FUNCTION_BLOCK fb_gm_measurementModule
VAR_INPUT
	SFCInit : BOOL;
END_VAR
VAR_OUTPUT
END_VAR
VAR
	trn_connectionCheckDone: BOOL;
	trn_wattingForLensDone: BOOL;
	flg_buf_gateLengthISSuccessed: BOOL;
	flg_buf_dummySignal: BOOL;
	trn_readCavDone: BOOL;
	fbi_getCav: fb_getCav;
	trn_chuckDone: BOOL;
	var_chuckCount: INT;
	trn_requestPickUpDone: BOOL;
	TON_data: TON;
	fbi_delayTimer: TON;
	trn_AddCountDone: BOOL;
	trn_lotStampDone: BOOL;
	var_process: INT;
	fbi_ton: TON;
	trn_LensCheckDone: BOOL;
	flg_SensorCheckDone: BOOL;
	flg_incjet_runned: BOOL;
END_VAR

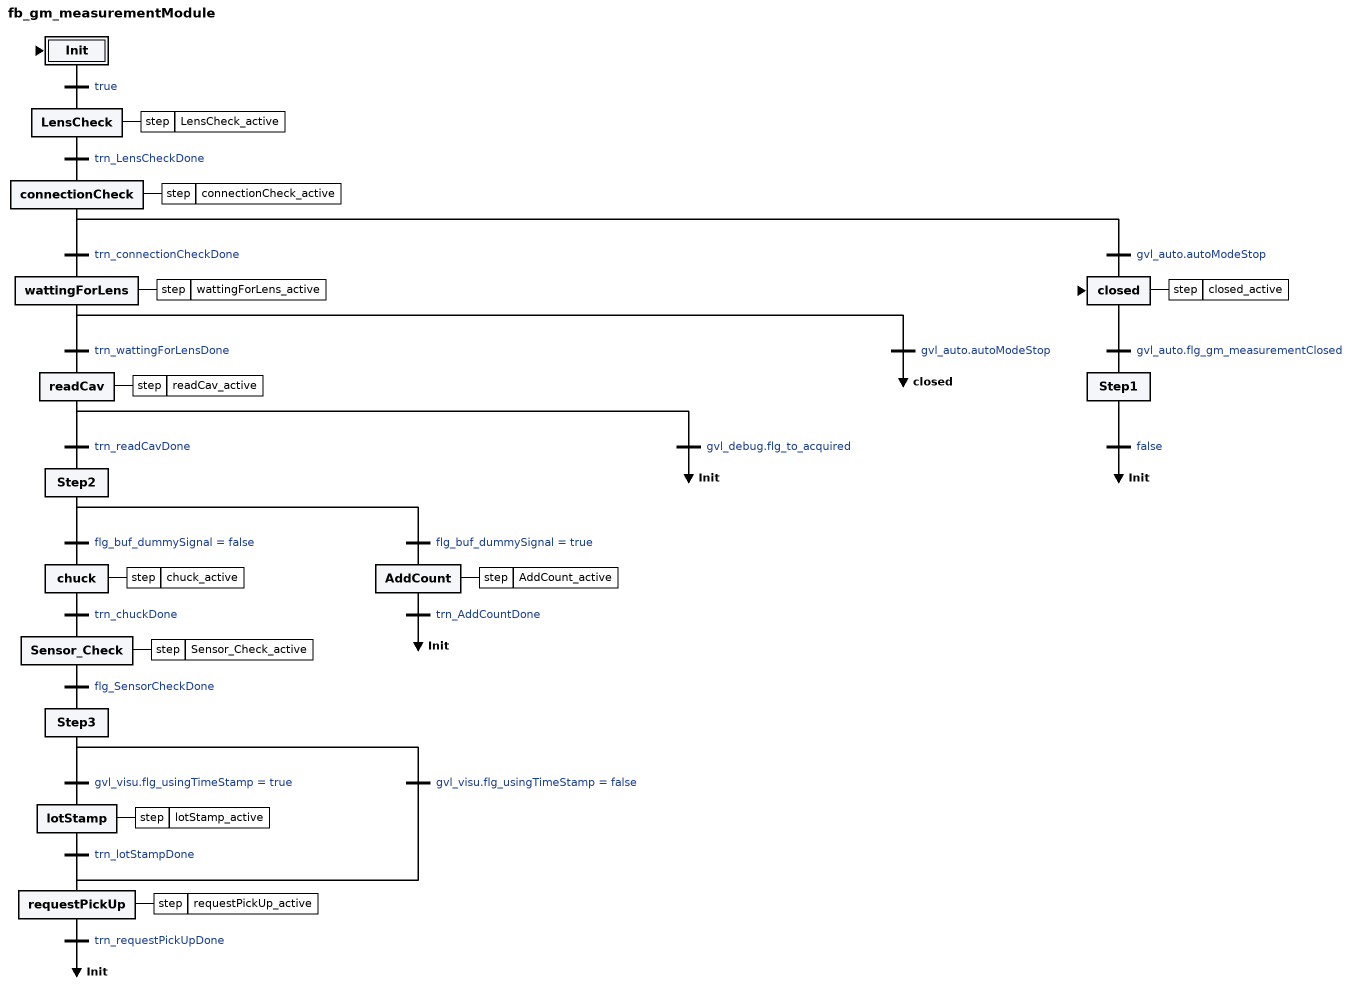
INITIAL_STEP Init:
END_STEP
TRANSITION FROM Init TO LensCheck
    := true;
END_TRANSITION
STEP LensCheck:
    LensCheck_active(N);  // step action
END_STEP
TRANSITION FROM LensCheck TO connectionCheck
    := trn_LensCheckDone;
END_TRANSITION
STEP connectionCheck:
    connectionCheck_active(N);  // step action
END_STEP
TRANSITION FROM connectionCheck TO wattingForLens
    := trn_connectionCheckDone;
END_TRANSITION
STEP wattingForLens:
    wattingForLens_active(N);  // step action
END_STEP
TRANSITION FROM wattingForLens TO readCav
    := trn_wattingForLensDone;
END_TRANSITION
TRANSITION FROM wattingForLens TO closed
    := gvl_auto.autoModeStop;
END_TRANSITION
TRANSITION FROM connectionCheck TO closed
    := gvl_auto.autoModeStop;
END_TRANSITION
STEP closed:
    closed_active(N);  // step action
END_STEP
TRANSITION FROM closed TO Step1
    := gvl_auto.flg_gm_measurementClosed;
END_TRANSITION
STEP Step1:
END_STEP
TRANSITION FROM Step1 TO Init
    := false;
END_TRANSITION
STEP readCav:
    readCav_active(N);  // step action
END_STEP
TRANSITION FROM readCav TO Step2
    := trn_readCavDone;
END_TRANSITION
TRANSITION FROM readCav TO Init
    := gvl_debug.flg_to_acquired;
END_TRANSITION
STEP Step2:
END_STEP
TRANSITION FROM Step2 TO chuck
    := flg_buf_dummySignal = false;
END_TRANSITION
TRANSITION FROM Step2 TO AddCount
    := flg_buf_dummySignal = true;
END_TRANSITION
STEP AddCount:
    AddCount_active(N);  // step action
END_STEP
TRANSITION FROM AddCount TO Init
    := trn_AddCountDone;
END_TRANSITION
STEP chuck:
    chuck_active(N);  // step action
END_STEP
TRANSITION FROM chuck TO Sensor_Check
    := trn_chuckDone;
END_TRANSITION
STEP Sensor_Check:
    Sensor_Check_active(N);  // step action
END_STEP
TRANSITION FROM Sensor_Check TO Step3
    := flg_SensorCheckDone;
END_TRANSITION
STEP Step3:
END_STEP
TRANSITION FROM Step3 TO lotStamp
    := gvl_visu.flg_usingTimeStamp = true;
END_TRANSITION
STEP lotStamp:
    lotStamp_active(N);  // step action
END_STEP
TRANSITION FROM lotStamp TO requestPickUp
    := trn_lotStampDone;
END_TRANSITION
TRANSITION FROM Step3 TO requestPickUp
    := gvl_visu.flg_usingTimeStamp = false;
END_TRANSITION
STEP requestPickUp:
    requestPickUp_active(N);  // step action
END_STEP
TRANSITION FROM requestPickUp TO Init
    := trn_requestPickUpDone;
END_TRANSITION

ACTION AddCount_active:
IF AddCount._x AND AddCount.x = FALSE THEN
	trn_AddCountDone := FALSE;
ELSIF AddCount._x AND AddCount.x THEN
	IF gvl_visu.flg_missingParts THEN
		gvl_gm.var_buf_measurementCav := gvl_auto.pocketNo[gvl_auto.buf_cavNo] + 1;
		trn_AddCountDone := TRUE;
	ELSE
		trn_AddCountDone := TRUE;
	END_IF
END_IF
END_ACTION

ACTION chuck_active:
IF chuck._x AND chuck.x = FALSE THEN
	TON_data.IN := FALSE;;
	trn_chuckDone := FALSE;
	gvl_solv.fbi_gm_chuck.in_flg_run := FALSE;
	gvl_solv.fbi_gm_push.in_flg_run := FALSE;
	gvl_auto.flg_gateData_Tx := FALSE;
	var_chuckCount := -11;
ELSIF chuck._x AND chuck.x THEN
	CASE var_chuckCount OF
		-11:
			IF gvl_param.var_productInfo[gvl_param.var_currentProductID].flg_mode_measurement THEN
				var_chuckCount := -10;
			ELSE
				var_chuckCount := 0;
			END_IF
		-10:
			gvl_solv.fbi_gm_push.in_var_moveMode := eP_svMoveMode.svB;
			gvl_solv.fbi_gm_push.in_flg_run := TRUE;
			var_chuckCount := -9;
		-9:
			IF gvl_solv.fbi_gm_push.out_flg_Done THEN
				gvl_solv.fbi_gm_push.in_flg_run := FALSE;
				var_chuckCount := -8;
			END_IF
		-8:
			gvl_solv.fbi_gm_push.in_var_moveMode := eP_svMoveMode.svA;
			gvl_solv.fbi_gm_push.in_flg_run := TRUE;
			var_chuckCount := -7;
		-7:
			IF gvl_solv.fbi_gm_push.out_flg_Done THEN
				gvl_solv.fbi_gm_push.in_flg_run := FALSE;
				var_chuckCount := -6;
			END_IF
		-6:
			gvl_solv.fbi_gm_chuck.in_var_moveMode := eP_svMoveMode.svB;
			gvl_solv.fbi_gm_chuck.in_flg_run := TRUE;
			var_chuckCount := -5;
		-5:
			IF gvl_solv.fbi_gm_chuck.out_flg_Done THEN
				gvl_solv.fbi_gm_chuck.in_flg_run := FALSE;
				var_chuckCount := -4;
			END_IF
		-4:
			gvl_solv.fbi_gm_push.in_var_moveMode := eP_svMoveMode.svB;
			gvl_solv.fbi_gm_push.in_flg_run := TRUE;
			var_chuckCount := -3;
		-3:
			IF gvl_solv.fbi_gm_push.out_flg_Done THEN
				gvl_solv.fbi_gm_push.in_flg_run := FALSE;
				var_chuckCount := 6;
			END_IF
		0:
			gvl_solv.fbi_gm_chuck.in_var_moveMode := eP_svMoveMode.svB;
			gvl_solv.fbi_gm_chuck.in_flg_run := TRUE;
			var_chuckCount := 1;
		1:
			
			IF gvl_solv.fbi_gm_chuck.out_flg_Done THEN
				gvl_solv.fbi_gm_chuck.in_flg_run := FALSE;
				var_chuckCount := 2;
			END_IF
		2:
			
			gvl_solv.fbi_gm_chuck.in_var_moveMode := eP_svMoveMode.svA;
			gvl_solv.fbi_gm_push.in_var_moveMode := eP_svMoveMode.svB;
			gvl_solv.fbi_gm_push.in_flg_run := TRUE;
			gvl_solv.fbi_gm_chuck.in_flg_run := TRUE;
			var_chuckCount := 3;
		3:
			IF gvl_solv.fbi_gm_push.out_flg_Done THEN
				gvl_solv.fbi_gm_push.in_flg_run := FALSE;
				gvl_solv.fbi_gm_chuck.in_flg_run := FALSE;
				var_chuckCount := 4;
			END_IF
		4:
			gvl_solv.fbi_gm_chuck.in_var_moveMode := eP_svMoveMode.svB;
			gvl_solv.fbi_gm_chuck.in_flg_run := TRUE;
			var_chuckCount := 5;
		5:
			IF gvl_solv.fbi_gm_chuck.out_flg_Done THEN
				gvl_solv.fbi_gm_chuck.in_flg_run := FALSE;
				var_chuckCount := 6;
			END_IF
		6:	
			TON_data.IN := TRUE;
			IF TON_data.Q THEN
				var_chuckCount := 7;
			END_IF
		7://gate measurement
			TON_data.IN := FALSE;
			IF gvl_io.flg_gm_fiberSens AND (gvl_io.var_gateLength > gvl_param.var_productInfo[gvl_param.var_currentProductID].gateLength_max OR gvl_io.var_gateLength < gvl_param.var_productInfo[gvl_param.var_currentProductID].gateLength_min) THEN
				gvl_gm.flg_gateLengthIsPassed := FALSE;
			ELSE
				gvl_gm.flg_gateLengthIsPassed := TRUE;
			END_IF
			gvl_auto.flg_gateData_Tx := TRUE;
			var_chuckCount := 8;
		8:
			gvl_solv.fbi_gm_chuck.in_flg_run := FALSE;
			var_chuckCount := 9;
		9:
			trn_chuckDone := TRUE;
	END_CASE
END_IF
TON_data(IN:= , PT:=T#200MS , Q=> , ET=> );
END_ACTION

ACTION closed_active:
IF closed._x AND closed.x = FALSE THEN
	gvl_auto.flg_gm_measurementClosed := FALSE;
ELSIF closed._x AND closed.x THEN
	gvl_io.flg_requestLens := FALSE;
	gvl_auto.flg_gm_measurementClosed := TRUE;
END_IF
END_ACTION

ACTION connectionCheck_active:
IF connectionCheck._x AND connectionCheck.x = FALSE THEN
	trn_connectionCheckDone:= FALSE;
	gvl_io.flg_requestLens := TRUE;
	var_process := 0;
ELSIF connectionCheck._x AND connectionCheck.x THEN
	CASE var_process OF
		0:
			IF gvl_io.flg_bitNumber0 
				AND gvl_io.flg_bitNumber1
				AND gvl_io.flg_bitNumber2
				AND gvl_io.flg_bitNumber3 OR gvl_debug.cavConecctSkip THEN
				trn_connectionCheckDone:= TRUE;
			END_IF
			IF NOT gvl_visu.flg_btn_vacSensOn THEN
				IF gvl_io.flg_gm_fiberSens THEN
					gvl_io.flg_requestLens := FALSE;
					IF((gvl_axis.axisX.NcToPlc.ActPos < gvl_visu.var_in_initialPos.x + 1) AND (gvl_axis.axisX.NcToPlc.ActPos > gvl_visu.var_in_initialPos.x - 1) AND NOT gvl_io.flg_fiberSens AND gvl_io.out_wire_ejectorVac ) THEN
						gvl_error.flg_gm_fiberSens := TRUE;
					END_IF
				END_IF
			END_IF
	END_CASE
	
END_IF
END_ACTION

ACTION LensCheck_active:
IF LensCheck._x AND LensCheck.x = FALSE THEN
	trn_LensCheckDone := FALSE;
	gvl_debug.flg_to_demand:= FALSE;
ELSIF LensCheck._x AND LensCheck.x THEN
	IF gvl_debug.out_busy THEN
		trn_LensCheckDone := TRUE;
	ELSE
		IF gvl_io.flg_gm_fiberSens THEN
			gvl_error.flg_gm_fiberSens := TRUE;	
		ELSE
			trn_LensCheckDone := TRUE;
		END_IF	
	END_IF
END_IF
END_ACTION

ACTION lotStamp_active:
IF lotStamp._x AND lotStamp.x = FALSE THEN
	trn_lotStampDone := FALSE;
	var_process := 0;
	fbi_ton.IN := FALSE;
	flg_incjet_runned:= FALSE;
ELSIF lotStamp._x AND lotStamp.x THEN
	CASE var_process OF
		0:
			fbi_ton.PT:= T#5S;
			fbi_ton.IN := TRUE;
			gvl_error.flg_incjet := fbi_ton.Q;
			gvl_gm.var_incjetInfo.flg_denyStamp := gvl_io.flg_gm_fiberSens;
			IF gvl_gm.var_incjetInfo.flg_stampReady THEN
				var_process := 1;
			END_IF
		1:
			fbi_ton.IN := FALSE;
			gvl_solv.fbi_gm_stamp.in_flg_run := FALSE;
			gvl_solv.fbi_gm_stamp.in_var_moveMode := eP_svMoveMode.svB;
			var_process := 2;
			
		2:
			gvl_solv.fbi_gm_stamp.in_flg_run := TRUE;
			var_process := 3;
		3:
			IF gvl_gm.var_incjetInfo.flg_stampRun THEN
				flg_incjet_runned:= TRUE;
			END_IF
			IF gvl_solv.fbi_gm_stamp.out_flg_Done THEN
				gvl_solv.fbi_gm_stamp.in_flg_run := FALSE;
				var_process := 4;
			END_IF
		4:
			fbi_ton.PT:= T#0.2S;
			fbi_ton.IN := TRUE;
			IF gvl_gm.var_incjetInfo.flg_stampRun THEN
				flg_incjet_runned:= TRUE;
			END_IF
			IF fbi_ton.Q THEN
				var_process := 5;
			END_IF
		5:
			IF flg_incjet_runned OR NOT gvl_gm.var_incjetInfo.flg_denyStamp THEN
				var_process := 6;
			ELSE
				gvl_error.flg_incjet:= TRUE;
			END_IF
		6:
			fbi_ton.IN := FALSE;
			gvl_solv.fbi_gm_stamp.in_var_moveMode := eP_svMoveMode.svA;
			gvl_solv.fbi_gm_stamp.in_flg_run := TRUE;
			var_process := 7;
		7:
			IF gvl_solv.fbi_gm_stamp.out_flg_Done THEN
				gvl_solv.fbi_gm_stamp.in_flg_run := FALSE;
				var_process := 8;
			END_IF
		8:
			flg_incjet_runned:= FALSE;
			gvl_gm.var_incjetInfo.flg_denyStamp := FALSE;
			trn_lotStampDone := TRUE;
	END_CASE
END_IF
fbi_ton(IN:= , PT:= , Q=> , ET=> );
END_ACTION

ACTION readCav_active:
IF readCav._x AND readCav.x = FALSE THEN
	trn_readCavDone := FALSE;
	THIS^.fbi_getCav();
	fbi_getCav.in_flg_run := FALSE;
	fbi_delayTimer.IN := FALSE;
ELSIF readCav._x AND readCav.x THEN
	THIS^.fbi_getCav();
	fbi_delayTimer.IN := TRUE;
	THIS^.fbi_getCav.in_flg_run := fbi_delayTimer.Q;
	IF gvl_debug.flg_debug_run THEN
		gvl_gm.var_buf_measurementCav := gvl_debug.var_cav;
		IF NOT (gvl_debug.flg_check_quality AND gvl_debug.flg_to_measurement) THEN
			trn_readCavDone := TRUE;
		END_IF
	ELSE
		IF THIS^.fbi_getCav.out_flg_Done THEN
			gvl_gm.var_buf_measurementCav := THIS^.fbi_getCav.out_var_cav;
			IF gvl_debug.flg_check_quality AND gvl_debug.flg_to_measurement THEN
				gvl_debug.flg_to_demand:= TRUE;
			ELSE
				trn_readCavDone := TRUE;
			END_IF
		ELSIF THIS^.fbi_getCav.out_flg_error THEN
			gvl_auto.cavNo := 0;
			IF gvl_debug.flg_check_quality AND gvl_debug.flg_to_measurement THEN
				gvl_debug.flg_to_demand:= TRUE;
			ELSE
				trn_readCavDone := TRUE;
			END_IF
		END_IF
	END_IF	
	
END_IF
fbi_delayTimer(IN:= , PT:=T#100MS , Q=> , ET=> );
END_ACTION

ACTION requestPickUp_active:
IF requestPickUp._x AND requestPickUp.x = FALSE THEN
	gvl_gm.flg_lensPickUpDone := FALSE;
	gvl_gm.flg_requestPickup := FALSE;
	trn_requestPickUpDone := false;
ELSIF requestPickUp._x AND requestPickUp.x THEN
	IF gvl_gm.flg_lensPickUpDone THEN
		gvl_gm.flg_requestPickup := FALSE;
		trn_requestPickUpDone := TRUE;
	ELSE
		gvl_gm.flg_requestPickup := TRUE;
	END_IF
END_IF
END_ACTION

ACTION Sensor_Check_active:
IF Sensor_Check._x AND Sensor_Check.x = FALSE THEN
	flg_SensorCheckDone := FALSE;
ELSIF Sensor_Check._x AND Sensor_Check.x THEN
	IF gvl_visu.flg_btn_vacSensOn THEN
		flg_SensorCheckDone:= TRUE;
	ELSE
		IF gvl_io.flg_gm_fiberSens THEN
			flg_SensorCheckDone:= TRUE;
		ELSE
			IF((gvl_axis.axisX.NcToPlc.ActPos < gvl_visu.var_in_initialPos.x + 1) AND (gvl_axis.axisX.NcToPlc.ActPos > gvl_visu.var_in_initialPos.x - 1) AND NOT gvl_io.flg_fiberSens AND gvl_io.out_wire_ejectorVac ) THEN
				gvl_error.flg_gm_fiberSens := TRUE;
			END_IF
		END_IF
	END_IF
END_IF
END_ACTION

ACTION wattingForLens_active:
IF wattingForLens._x AND wattingForLens.x = FALSE THEN
	trn_wattingForLensDone := FALSE;
	flg_buf_gateLengthISSuccessed := FALSE;
	flg_buf_dummySignal := FALSE;
ELSIF wattingForLens._x AND wattingForLens.x THEN
	//gate
	IF gvl_IO.flg_gateLengthIsSuccessed  THEN
		flg_buf_gateLengthISSuccessed := TRUE;
	END_IF
	//dummy signal
	IF gvl_io.flg_dummySiganl THEN
		flg_buf_dummySignal := TRUE;
	END_IF
	//lens set done
	IF gvl_debug.out_busy THEN
		IF gvl_visu.flg_btn_lensSetDone OR gvl_visu.flg_btn_vacSensOn THEN
			gvl_io.flg_requestLens := FALSE;
			trn_wattingForLensDone := TRUE;
		END_IF
	ELSE
		IF gvl_io.flg_lensSetDone THEN
			gvl_io.flg_requestLens := FALSE; 
			trn_wattingForLensDone := TRUE;
		END_IF
	END_IF
END_IF
END_ACTION

END_FUNCTION_BLOCK

(* stored: Version 1.1.0.1, ProductVersion 3.1.4024.11
   POU fb_gm_measurementModule: Id {e564b2af-f26e-465c-8cfd-522f40911ebd}, SpecialFunc None
   Action AddCount_active: Id {c657e98d-1a60-46c8-b7d6-e66e6ef44e71}
   Action chuck_active: Id {6b24fa23-7c1a-4114-905e-25f3a8212f6b}
   Action closed_active: Id {0aba8fe8-323a-417a-baaf-24601c409549}
   Action connectionCheck_active: Id {e834891a-b105-4590-ab4b-9e66393d31b6}
   Action LensCheck_active: Id {312bd6c4-31ea-4ac4-b036-c5edc7d077c5}
   Action lotStamp_active: Id {e67c0742-f1e2-42a6-b0bc-a02eaca34927}
   Action readCav_active: Id {4c82aff0-e11a-46c3-90c2-f6e725474125}
   Action requestPickUp_active: Id {f87796ec-d869-463e-b016-7c81db2cb043}
   Action Sensor_Check_active: Id {a7d8b61e-629d-4902-a021-4f2ac101c6f2}
   Action wattingForLens_active: Id {5f1f5772-dd55-4fd1-8af3-42c2f354edf0} *)
